RoboDK station: Stringer C-Top4-BOX1.rdk

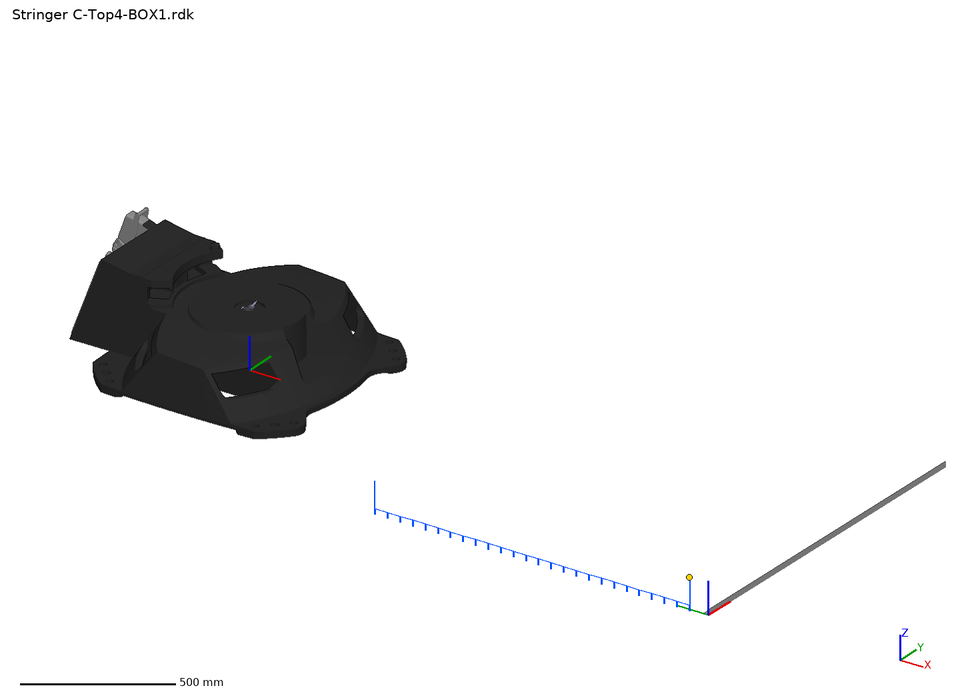
[picture v0: the station drawn from its stored meshes, robots at their saved joint values, targets as dots, program paths as lines]
Station Stringer C-Top4-BOX1 (saved by RoboDK 5.2.3). Poses are relative to the parent item; angles as X-Y-Z fixed-axis rotations.
  - frame KUKA KR 210 R2700 extra Base at (0, 0, 0) mm
    - robot KUKA KR 210 R2700 extra: 6 axes, payload 210 kg, reach 2696 mm, repeatability 0.06 mm, weight 1068 kg
        joint limits [-185, -140, -120, -350, -125, -350] to [185, -5, 155, 350, 125, 350]; home [0, -90, 90, 0, 0, 0]; saved at [-38.394, -22.339, 84.746, 101.478, 23.35, -134.058]
      - tool Spindle, TCP at (32, 0, 260) mm, rotated rx 0 ry 39 rz 0 deg, size 157.3 x 72 x 259.9 mm
  - frame Frame 2 at (1800, 0, -372.68) mm, rotated rx 0 ry 0 rz 90 deg
    - object L-Stringer C - Top4-BOX1 at (0, 0, 0) mm, size 1324.9 x 20 x 20 mm, geometry from L-Stringer C - Top4-BOX1.stl
    - object Stringer C-Top4-BOX1 at (0, 0, 0) mm, rotated rx 0 ry 0 rz -90 deg, 26 curves, geometry from Point 26
  - machining project Point settings: rotZ(0) | rotX(0)*rotY(0) | rotz(0) | onStart | onPathStart | onApproach | onPoint | onRetract | onFinish | SetRPM(%1) | SetTool(%1) | Extruder(%1) | default | default | OutOnMov(%1) | OutOffMov(%1) | onPathFinish | M_RunCode(%1)
  - program Point (141 instructions, listed below)
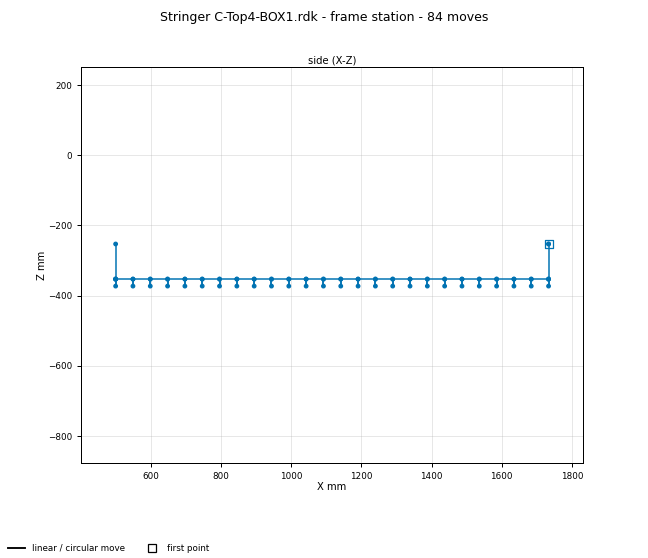
[picture p0: tool path of Stringer C-Top4-BOX1.rdk in frame station, 84 of 84 moves have a stored position in this frame; points joined in program order, loops and branches not executed]

--- program Point (robot KUKA KR 210 R2700 extra) ---
  Smooth(1)
  Set speed (1000.0 mm/s)
  Set Ref.: Frame 2
  Set Tool: Spindle
  Show Spindle
  MoveJ 1 to (-10.8, 66.57, 120) mm, rotated rx -180 ry 0 rz -180 deg; joints [-2.516, -34.008, 111.818, 176.491, 26.827, -178.823]
  MoveL 2 to (-10.8, 66.57, 120) mm, rotated rx -180 ry 0 rz -180 deg; joints [-2.516, -34.008, 111.818, 176.491, 26.827, -178.823]
  MoveL 3 to (-10.8, 66.57, 20) mm, rotated rx 180 ry 0 rz 180 deg; joints [-2.516, -28.68, 109.176, 176.785, 29.508, -179.157]
  MoveL 4 to (-10.8, 66.57, 20) mm, rotated rx 180 ry 0 rz 180 deg; joints [-2.516, -28.68, 109.176, 176.785, 29.508, -179.157]
  Set speed (50.0 mm/s)
  MoveL 5 to (-10.8, 66.57, 0) mm, rotated rx 180 ry 0 rz -180 deg; joints [-2.516, -27.622, 108.601, 176.832, 29.989, -179.211]
  MoveL 6 to (-10.8, 66.57, 20) mm, rotated rx 180 ry 0 rz 180 deg; joints [-2.516, -28.68, 109.176, 176.785, 29.508, -179.157]
  Set speed (1000.0 mm/s)
  MoveL 7 to (-10.8, 115.91, 20) mm, rotated rx -180 ry 0 rz -180 deg; joints [-4.375, -28.659, 109.022, 174.388, 29.399, -178.51]
  Set speed (50.0 mm/s)
  MoveL 8 to (-10.8, 115.91, 0) mm, rotated rx -180 ry 0 rz -180 deg; joints [-4.375, -27.603, 108.447, 174.47, 29.878, -178.604]
  MoveL 9 to (-10.8, 115.91, 20) mm, rotated rx -180 ry 0 rz -180 deg; joints [-4.375, -28.659, 109.022, 174.388, 29.399, -178.51]
  Set speed (1000.0 mm/s)
  MoveL 10 to (-10.8, 165.24, 20) mm, rotated rx 180 ry 0 rz 180 deg; joints [-6.224, -28.626, 108.785, 171.969, 29.234, -177.826]
  Set speed (50.0 mm/s)
  MoveL 11 to (-10.8, 165.24, 0) mm, rotated rx -180 ry 0 rz -180 deg; joints [-6.224, -27.572, 108.211, 172.087, 29.709, -177.961]
  MoveL 12 to (-10.8, 165.24, 20) mm, rotated rx 180 ry 0 rz 180 deg; joints [-6.224, -28.626, 108.785, 171.969, 29.234, -177.826]
  Set speed (1000.0 mm/s)
  MoveL 13 to (-10.8, 214.58, 20) mm, rotated rx -180 ry 0 rz -180 deg; joints [-8.061, -28.58, 108.465, 169.517, 29.014, -177.09]
  Set speed (50.0 mm/s)
  MoveL 14 to (-10.8, 214.58, 0) mm, rotated rx -180 ry 0 rz -180 deg; joints [-8.061, -27.529, 107.892, 169.671, 29.484, -177.266]
  MoveL 15 to (-10.8, 214.58, 20) mm, rotated rx -180 ry 0 rz -180 deg; joints [-8.061, -28.58, 108.465, 169.517, 29.014, -177.09]
  Set speed (1000.0 mm/s)
  MoveL 16 to (-10.8, 263.92, 20) mm, rotated rx -180 ry 0 rz -180 deg; joints [-9.881, -28.521, 108.062, 167.022, 28.744, -176.286]
  Set speed (50.0 mm/s)
  MoveL 17 to (-10.8, 263.92, 0) mm, rotated rx 180 ry 0 rz 180 deg; joints [-9.881, -27.474, 107.491, 167.214, 29.208, -176.505]
  MoveL 18 to (-10.8, 263.92, 20) mm, rotated rx -180 ry 0 rz -180 deg; joints [-9.881, -28.521, 108.062, 167.022, 28.744, -176.286]
  Set speed (1000.0 mm/s)
  MoveL 19 to (-10.8, 313.25, 20) mm, rotated rx 180 ry 0 rz 180 deg; joints [-11.681, -28.447, 107.577, 164.475, 28.427, -175.399]
  Set speed (50.0 mm/s)
  MoveL 20 to (-10.8, 313.25, 0) mm, rotated rx 180 ry 0 rz -180 deg; joints [-11.681, -27.404, 107.007, 164.705, 28.883, -175.662]
  MoveL 21 to (-10.8, 313.25, 20) mm, rotated rx 180 ry 0 rz 180 deg; joints [-11.681, -28.447, 107.577, 164.475, 28.427, -175.399]
  Set speed (1000.0 mm/s)
  MoveL 22 to (-10.8, 362.59, 20) mm, rotated rx -180 ry 0 rz -180 deg; joints [-13.458, -28.357, 107.009, 161.864, 28.069, -174.415]
  Set speed (50.0 mm/s)
  MoveL 23 to (-10.8, 362.59, 0) mm, rotated rx 180 ry 0 rz 180 deg; joints [-13.458, -27.319, 106.441, 162.134, 28.517, -174.722]
  MoveL 24 to (-10.8, 362.59, 20) mm, rotated rx -180 ry 0 rz -180 deg; joints [-13.458, -28.357, 107.009, 161.864, 28.069, -174.415]
  Set speed (1000.0 mm/s)
  MoveL 25 to (-10.8, 411.92, 20) mm, rotated rx -180 ry 0 rz -180 deg; joints [-15.209, -28.249, 106.36, 159.179, 27.676, -173.318]
  Set speed (50.0 mm/s)
  MoveL 26 to (-10.8, 411.92, 0) mm, rotated rx 180 ry 0 rz 180 deg; joints [-15.209, -27.216, 105.794, 159.49, 28.113, -173.67]
  MoveL 27 to (-10.8, 411.92, 20) mm, rotated rx -180 ry 0 rz -180 deg; joints [-15.209, -28.249, 106.36, 159.179, 27.676, -173.318]
  Set speed (1000.0 mm/s)
  MoveL 28 to (-10.8, 461.26, 20) mm, rotated rx 180 ry 0 rz -180 deg; joints [-16.932, -28.122, 105.629, 156.408, 27.255, -172.092]
  Set speed (50.0 mm/s)
  MoveL 29 to (-10.8, 461.26, 0) mm, rotated rx 180 ry 0 rz 180 deg; joints [-16.932, -27.095, 105.065, 156.762, 27.68, -172.492]
  MoveL 30 to (-10.8, 461.26, 20) mm, rotated rx 180 ry 0 rz -180 deg; joints [-16.932, -28.122, 105.629, 156.408, 27.255, -172.092]
  Set speed (1000.0 mm/s)
  MoveL 31 to (-10.8, 510.6, 20) mm, rotated rx 180 ry 0 rz 180 deg; joints [-18.624, -27.974, 104.817, 153.541, 26.812, -170.726]
  Set speed (50.0 mm/s)
  MoveL 32 to (-10.8, 510.6, 0) mm, rotated rx -180 ry 0 rz -180 deg; joints [-18.624, -26.954, 104.255, 153.939, 27.223, -171.173]
  MoveL 33 to (-10.8, 510.6, 20) mm, rotated rx 180 ry 0 rz 180 deg; joints [-18.624, -27.974, 104.817, 153.541, 26.812, -170.726]
  Set speed (1000.0 mm/s)
  MoveL 34 to (-10.8, 559.93, 20) mm, rotated rx 180 ry 0 rz 180 deg; joints [-20.282, -27.803, 103.924, 150.568, 26.355, -169.204]
  Set speed (50.0 mm/s)
  MoveL 35 to (-10.8, 559.93, 0) mm, rotated rx 180 ry 0 rz 180 deg; joints [-20.282, -26.79, 103.365, 151.011, 26.752, -169.7]
  MoveL 36 to (-10.8, 559.93, 20) mm, rotated rx 180 ry 0 rz 180 deg; joints [-20.282, -27.803, 103.924, 150.568, 26.355, -169.204]
  Set speed (1000.0 mm/s)
  MoveL 37 to (-10.8, 609.27, 20) mm, rotated rx 180 ry 0 rz 180 deg; joints [-21.906, -27.607, 102.95, 147.477, 25.894, -167.515]
  Set speed (50.0 mm/s)
  MoveL 38 to (-10.8, 609.27, 0) mm, rotated rx 180 ry 0 rz -180 deg; joints [-21.906, -26.602, 102.393, 147.968, 26.274, -168.061]
  MoveL 39 to (-10.8, 609.27, 20) mm, rotated rx 180 ry 0 rz 180 deg; joints [-21.906, -27.607, 102.95, 147.477, 25.894, -167.515]
  Set speed (1000.0 mm/s)
  MoveL 40 to (-10.8, 658.6, 20) mm, rotated rx -180 ry 0 rz -180 deg; joints [-23.494, -27.385, 101.895, 144.262, 25.437, -165.649]
  Set speed (50.0 mm/s)
  MoveL 41 to (-10.8, 658.6, 0) mm, rotated rx -180 ry 0 rz -180 deg; joints [-23.494, -26.388, 101.342, 144.799, 25.799, -166.245]
  MoveL 42 to (-10.8, 658.6, 20) mm, rotated rx -180 ry 0 rz -180 deg; joints [-23.494, -27.385, 101.895, 144.262, 25.437, -165.649]
  Set speed (1000.0 mm/s)
  MoveL 43 to (-10.8, 707.94, 20) mm, rotated rx -180 ry 0 rz -180 deg; joints [-25.044, -27.134, 100.761, 140.913, 24.994, -163.595]
  Set speed (50.0 mm/s)
  MoveL 44 to (-10.8, 707.94, 0) mm, rotated rx -180 ry 0 rz -180 deg; joints [-25.044, -26.145, 100.21, 141.497, 25.335, -164.24]
  MoveL 45 to (-10.8, 707.94, 20) mm, rotated rx -180 ry 0 rz -180 deg; joints [-25.044, -27.134, 100.761, 140.913, 24.994, -163.595]
  Set speed (1000.0 mm/s)
  MoveL 46 to (-10.8, 757.28, 20) mm, rotated rx 180 ry 0 rz 180 deg; joints [-26.556, -26.853, 99.546, 137.425, 24.573, -161.347]
  Set speed (50.0 mm/s)
  MoveL 47 to (-10.8, 757.28, 0) mm, rotated rx 180 ry 0 rz -180 deg; joints [-26.556, -25.873, 98.997, 138.055, 24.893, -162.042]
  MoveL 48 to (-10.8, 757.28, 20) mm, rotated rx 180 ry 0 rz 180 deg; joints [-26.556, -26.853, 99.546, 137.425, 24.573, -161.347]
  Set speed (1000.0 mm/s)
  MoveL 49 to (-10.8, 806.61, 20) mm, rotated rx -180 ry 0 rz -180 deg; joints [-28.029, -26.54, 98.25, 133.796, 24.187, -158.903]
  Set speed (50.0 mm/s)
  MoveL 50 to (-10.8, 806.61, 0) mm, rotated rx 180 ry 0 rz -180 deg; joints [-28.029, -25.568, 97.704, 134.471, 24.483, -159.645]
  MoveL 51 to (-10.8, 806.61, 20) mm, rotated rx -180 ry 0 rz -180 deg; joints [-28.029, -26.54, 98.25, 133.796, 24.187, -158.903]
  Set speed (1000.0 mm/s)
  MoveL 52 to (-10.8, 855.95, 20) mm, rotated rx 180 ry 0 rz 180 deg; joints [-29.463, -26.193, 96.874, 130.027, 23.843, -156.264]
  Set speed (50.0 mm/s)
  MoveL 53 to (-10.8, 855.95, 0) mm, rotated rx 180 ry 0 rz -180 deg; joints [-29.463, -25.23, 96.33, 130.744, 24.115, -157.048]
  MoveL 54 to (-10.8, 855.95, 20) mm, rotated rx 180 ry 0 rz 180 deg; joints [-29.463, -26.193, 96.874, 130.027, 23.843, -156.264]
  Set speed (1000.0 mm/s)
  MoveL 55 to (-10.8, 905.28, 20) mm, rotated rx 180 ry 0 rz 180 deg; joints [-30.858, -25.809, 95.417, 126.124, 23.554, -153.434]
  Set speed (50.0 mm/s)
  MoveL 56 to (-10.8, 905.28, 0) mm, rotated rx -180 ry 0 rz -180 deg; joints [-30.858, -24.855, 94.875, 126.878, 23.799, -154.257]
  MoveL 57 to (-10.8, 905.28, 20) mm, rotated rx 180 ry 0 rz 180 deg; joints [-30.858, -25.809, 95.417, 126.124, 23.554, -153.434]
  Set speed (1000.0 mm/s)
  MoveL 58 to (-10.8, 954.62, 20) mm, rotated rx -180 ry 0 rz -180 deg; joints [-32.213, -25.388, 93.878, 122.096, 23.328, -150.423]
  Set speed (50.0 mm/s)
  MoveL 59 to (-10.8, 954.62, 0) mm, rotated rx 180 ry 0 rz 180 deg; joints [-32.213, -24.443, 93.337, 122.882, 23.545, -151.28]
  MoveL 60 to (-10.8, 954.62, 20) mm, rotated rx -180 ry 0 rz -180 deg; joints [-32.213, -25.388, 93.878, 122.096, 23.328, -150.423]
  Set speed (1000.0 mm/s)
  MoveL 61 to (-10.8, 1003.96, 20) mm, rotated rx -180 ry 0 rz -180 deg; joints [-33.529, -24.927, 92.255, 117.96, 23.176, -147.249]
  Set speed (50.0 mm/s)
  MoveL 62 to (-10.8, 1003.96, 0) mm, rotated rx 180 ry 0 rz -180 deg; joints [-33.529, -23.991, 91.716, 118.771, 23.364, -148.131]
  MoveL 63 to (-10.8, 1003.96, 20) mm, rotated rx -180 ry 0 rz -180 deg; joints [-33.529, -24.927, 92.255, 117.96, 23.176, -147.249]
  Set speed (1000.0 mm/s)
  MoveL 64 to (-10.8, 1053.29, 20) mm, rotated rx -180 ry 0 rz -180 deg; joints [-34.806, -24.424, 90.549, 113.738, 23.105, -143.933]
  Set speed (50.0 mm/s)
  MoveL 65 to (-10.8, 1053.29, 0) mm, rotated rx 180 ry 0 rz -180 deg; joints [-34.806, -23.498, 90.011, 114.564, 23.264, -144.832]
  MoveL 66 to (-10.8, 1053.29, 20) mm, rotated rx -180 ry 0 rz -180 deg; joints [-34.806, -24.424, 90.549, 113.738, 23.105, -143.933]
  Set speed (1000.0 mm/s)
  MoveL 67 to (-10.8, 1102.63, 20) mm, rotated rx 180 ry 0 rz 180 deg; joints [-36.045, -23.878, 88.757, 109.453, 23.124, -140.5]
  Set speed (50.0 mm/s)
  MoveL 68 to (-10.8, 1102.63, 0) mm, rotated rx -180 ry 0 rz -180 deg; joints [-36.045, -22.96, 88.219, 110.286, 23.253, -141.406]
  MoveL 69 to (-10.8, 1102.63, 20) mm, rotated rx 180 ry 0 rz 180 deg; joints [-36.045, -23.878, 88.757, 109.453, 23.124, -140.5]
  Set speed (1000.0 mm/s)
  MoveL 70 to (-10.8, 1151.96, 20) mm, rotated rx -180 ry 0 rz -180 deg; joints [-37.246, -23.286, 86.877, 105.138, 23.24, -136.982]
  Set speed (50.0 mm/s)
  MoveL 71 to (-10.8, 1151.96, 0) mm, rotated rx -180 ry 0 rz 180 deg; joints [-37.246, -22.377, 86.339, 105.967, 23.339, -137.885]
  MoveL 72 to (-10.8, 1151.96, 20) mm, rotated rx -180 ry 0 rz -180 deg; joints [-37.246, -23.286, 86.877, 105.138, 23.24, -136.982]
  Set speed (1000.0 mm/s)
  MoveL 73 to (-10.8, 1201.3, 20) mm, rotated rx -180 ry 0 rz -180 deg; joints [-38.41, -22.645, 84.906, 100.822, 23.457, -133.41]
  Set speed (50.0 mm/s)
  MoveL 74 to (-10.8, 1201.3, 0) mm, rotated rx -180 ry 0 rz -180 deg; joints [-38.41, -21.745, 84.367, 101.637, 23.527, -134.299]
  MoveL 75 to (-10.8, 1201.3, 20) mm, rotated rx -180 ry 0 rz -180 deg; joints [-38.41, -22.645, 84.906, 100.822, 23.457, -133.41]
  Set speed (1000.0 mm/s)
  MoveL 76 to (-10.8, 1250.64, 20) mm, rotated rx 180 ry 0 rz -180 deg; joints [-39.537, -21.954, 82.841, 96.538, 23.781, -129.818]
  Set speed (50.0 mm/s)
  MoveL 77 to (-10.8, 1250.64, 0) mm, rotated rx 180 ry 0 rz 180 deg; joints [-39.537, -21.062, 82.301, 97.329, 23.823, -130.683]
  MoveL 78 to (-10.8, 1250.64, 20) mm, rotated rx 180 ry 0 rz -180 deg; joints [-39.537, -21.954, 82.841, 96.538, 23.781, -129.818]
  Set speed (1000.0 mm/s)
  MoveL 79 to (-10.8, 1299.97, 20) mm, rotated rx -180 ry 0 rz -180 deg; joints [-40.629, -21.21, 80.679, 92.32, 24.213, -126.238]
  Set speed (50.0 mm/s)
  MoveL 80 to (-10.8, 1299.97, 0) mm, rotated rx -180 ry 0 rz -180 deg; joints [-40.629, -20.326, 80.136, 93.078, 24.229, -127.07]
  MoveL 81 to (-10.8, 1299.97, 20) mm, rotated rx -180 ry 0 rz -180 deg; joints [-40.629, -21.21, 80.679, 92.32, 24.213, -126.238]
  MoveL 82 to (-10.8, 1299.97, 20) mm, rotated rx -180 ry 0 rz -180 deg; joints [-40.629, -21.21, 80.679, 92.32, 24.213, -126.238]
  Set speed (1000.0 mm/s)
  MoveL 83 to (-10.8, 1299.97, 20) mm, rotated rx -180 ry 0 rz -180 deg; joints [-40.629, -21.21, 80.679, 92.32, 24.213, -126.238]
  MoveL 84 to (-10.8, 1299.97, 120) mm, rotated rx -180 ry 0 rz -180 deg; joints [-40.629, -25.571, 83.135, 88.081, 24.206, -121.591]
